FUNCTION_BLOCK Thermostat
VAR_INPUT
END_VAR
VAR_OUTPUT
END_VAR
VAR
	wInputAddress AT %I* : WORD;
	rScaleMax : REAL;
	rScaleMin : REAL;
	iTemperatureAnalogValue : INT;
	rTemperatureScaledValue : REAL;
END_VAR

METHOD FB_init : BOOL
VAR_INPUT
	bInitRetains : BOOL; // if TRUE, the retain variables are initialized (warm start / cold start)
	bInCopyCode : BOOL;  // if TRUE, the instance afterwards gets moved into the copy code (online change)
END_VAR
END_METHOD

METHOD PRIVATE scaleTemperature : REAL
VAR_INPUT
END_VAR
END_METHOD

PROPERTY PUBLIC temperature : REAL
GET
temperature := rTemperatureScaledValue;
END_GET
END_PROPERTY

END_FUNCTION_BLOCK

(* stored: Version 1.1.0.1, ProductVersion 3.1.4024.12
   POU Thermostat: Id {b2747955-fbbb-4ba2-b308-d456b12914c6}, SpecialFunc None
   Method FB_init: Id {5f7a32b8-7fa6-441f-a003-be979df5ffa4}
   Method scaleTemperature: Id {2ac7f04b-b036-498d-aa7d-5764fb1b441e}
   Property temperature: Id {08d80838-4a9e-468d-b957-bb1630d6392a}
   Get Get: Id {561e8b08-3d1f-4449-b269-db917a5ffd37} *)
